Staubli VAL3: sendData.pgx

public program sendData(sio& x_sSioSocket, num& x_nSendData[], RobotStatus& x_rRobotStatus, FlagStatus& x_fDataStatus)
  local num l_nSendNum
begin

  //This program is used for sending the feedback data to the host ROS contorller.

  //call the encodeSendData function to encrypt the sent data
  call encodeSendData(x_nSendData,x_rRobotStatus)

  //send the encrypted data to the host ROS controller
  l_nSendNum=sioSet(x_sSioSocket,x_nSendData)
  if l_nSendNum==52
    x_fDataStatus.RosFlag=1
  else
    x_fDataStatus.RosFlag=-1
  endIf

end
